FUNCTION Restore : BOOL
VAR_INPUT
END_VAR
VAR
	MotorDirectionEnum: MovementDirection;	// for better clarity on the direction 0 and 1
	MovementEnum: Movement; // for better clarity on the ON/OFF movement of the motors
END_VAR
VAR_IN_OUT	// REFERENCES!
	Restored: BOOL;
	AUTOMATICPositionAuto: INT;
	AUTOMATICPositionCurrent: INT;
	AUTOMATICSafetyON: BOOL;
	AUTOMATICCurrentlyMoving: BOOL;
	IODirection: BOOL;	
	IOMotor: BOOL;
END_VAR

IF AUTOMATICPositionAuto - AUTOMATICPositionCurrent > 5 AND (NOT Restored) AND (NOT AUTOMATICSafetyON) THEN
	IODirection := (MotorDirectionEnum = MovementDirection.AwayFromSensor);
	AUTOMATICCurrentlyMoving := TRUE;
	IOMotor := (MovementEnum = Movement.ON);
	Restored := FALSE;
ELSIF AUTOMATICPositionCurrent - AUTOMATICPositionAuto > 5 AND (NOT Restored) AND (NOT AUTOMATICSafetyON) THEN
	IODirection := (MotorDirectionEnum = MovementDirection.TowardsSensor);
	AUTOMATICCurrentlyMoving := TRUE;
	IOMotor := (MovementEnum = Movement.ON);
	Restored := FALSE;
ELSE
	AUTOMATICCurrentlyMoving := FALSE;
	IOMotor := (MovementEnum = Movement.OFF);
	Restored := TRUE;
END_IF

Restore := Restored;
RETURN;	// Restored

END_FUNCTION

(* stored: Version 1.1.0.1, ProductVersion 3.1.4024.13
   POU Restore: Id {c35f155a-143d-4f41-9a6e-6178c1b6d0e2}, SpecialFunc None *)
